FUNCTION_BLOCK FB_HDData
VAR_INPUT
	
    Alm :    BOOL ;//报警
	Wait :BOOL ;//待机
	Run :BOOL ;//运行
	XL_Wait:BOOL ;//下料等待时间
	Query:BOOL;//时间查询
	

END_VAR
VAR_OUTPUT
		STTimedata:ARRAY[0..32] OF ST_Timedata_1;

END_VAR
VAR
	
	rRun : R_TRIG;
	rAlm : R_TRIG;
	rWait : R_TRIG;
	rXL_Wait : R_TRIG;
	
	fRun: F_TRIG;
	fAlm: F_TRIG;
	fWait: F_TRIG;
    delay:BOOL ;//延时
	TON_1: TON;
	i:INT;
	K: INT;
	J: BOOL;
END_VAR

VAR_IN_OUT
     date1:INT;//查询日期
END_VAR

K:=K+1;
	IF K>499THEN
		J:=TRUE;
		K:=0;
	ELSE
		J:=FALSE;
	END_IF




///////////////运行时间/////////////////
rRun(CLK:= J , Q=> );

IF rRun.Q  AND  Run THEN
	STTimedata[system.stTime.wDay].RunTime[system.stTime.wHour]:=STTimedata[system.stTime.wDay].RunTime[system.stTime.wHour]+1;
END_IF

IF STTimedata[system.stTime.wDay].RunTime[system.stTime.wHour]> 3600 THEN
	STTimedata[system.stTime.wDay].RunTime[system.stTime.wHour]:= 3600 ;
END_IF

//IF STTimedata[system.stTime.wDay].AlmTime[system.stTime.wHour]= 0 AND STTimedata[system.stTime.wDay].WaitTime[system.stTime.wHour]= 0  AND 
   // (STTimedata[system.stTime.wDay].RunTime[system.stTime.wHour]= 3585  OR  STTimedata[system.stTime.wDay].RunTime[system.stTime.wHour]= 3586 ) THEN
	//STTimedata[system.stTime.wDay].RunTime[system.stTime.wHour]:= 3600 ;
//END_IF


///////////////待机时间///////////////
rWait(CLK:=J , Q=> );

IF rWait.Q  AND Wait THEN
	STTimedata[system.stTime.wDay].WaitTime[system.stTime.wHour]:=STTimedata[system.stTime.wDay].WaitTime[system.stTime.wHour]+1;
END_IF

IF STTimedata[system.stTime.wDay].WaitTime[system.stTime.wHour]> 3600 THEN
	STTimedata[system.stTime.wDay].WaitTime[system.stTime.wHour]:= 3600 ;
END_IF

//IF STTimedata[system.stTime.wDay].RunTime[system.stTime.wHour]= 0 AND STTimedata[system.stTime.wDay].AlmTime[system.stTime.wHour]= 0  AND 
  //   (STTimedata[system.stTime.wDay].RunTime[system.stTime.wHour]= 3585  OR  STTimedata[system.stTime.wDay].RunTime[system.stTime.wHour]= 3586 )  THEN
//	STTimedata[system.stTime.wDay].WaitTime[system.stTime.wHour]:= 3600 ;
//END_IF


////////////////报警时间///////////////
rAlm(CLK:=J , Q=> );

IF rAlm.Q AND Alm THEN
	STTimedata[system.stTime.wDay].AlmTime[system.stTime.wHour]:=STTimedata[system.stTime.wDay].AlmTime[system.stTime.wHour]+1;
END_IF

IF STTimedata[system.stTime.wDay].AlmTime[system.stTime.wHour]> 3600 THEN
	STTimedata[system.stTime.wDay].AlmTime[system.stTime.wHour]:= 3600 ;
END_IF

//IF STTimedata[system.stTime.wDay].RunTime[system.stTime.wHour]= 0 AND STTimedata[system.stTime.wDay].WaitTime[system.stTime.wHour]= 0  AND
 ////   (STTimedata[system.stTime.wDay].RunTime[system.stTime.wHour]= 3585  OR  STTimedata[system.stTime.wDay].RunTime[system.stTime.wHour]= 3586 ) THEN
//	STTimedata[system.stTime.wDay].AlmTime[system.stTime.wHour]:= 3600 ;
//END_IF

////////////////下料等待托盘时间///////////////
rXL_Wait(CLK:=J, Q=> );

IF rXL_Wait.Q AND XL_Wait THEN
	STTimedata[system.stTime.wDay].XLWaitTime[system.stTime.wHour]:=STTimedata[system.stTime.wDay].XLWaitTime[system.stTime.wHour]+1;
END_IF

//数据查询
IF Query THEN
	delay:=TRUE;
END_IF

TON_1(IN:= , PT:=T#60S , Q=> , ET=> );
IF delay THEN
		  IF NOT TON_1.Q THEN
			  TON_1.IN:=TRUE;
		  ELSE	
			  delay:=FALSE;
			  date1:=system.stTime.wDay;
		  END_IF	 
ELSE	
	 TON_1.IN:=FALSE;
END_IF


IF NOT delay THEN
STTimedata[32]:=STTimedata[system.stTime.wDay];
ELSE
STTimedata[32]:=STTimedata[date1];
END_IF

//数据清零
IF (system.stTime.wMonth=2 AND  system.stTime.wDay=28 )   OR
    ((system.stTime.wMonth=4 OR system.stTime.wMonth=6 OR system.stTime.wMonth=9 OR system.stTime.wMonth=11) AND system.stTime.wDay=30 )   OR
	((system.stTime.wMonth=1 OR  system.stTime.wMonth=3 OR system.stTime.wMonth=5 OR system.stTime.wMonth=7 OR system.stTime.wMonth=8 OR system.stTime.wMonth=10 OR system.stTime.wMonth=12) AND  system.stTime.wDay=31)  AND
    system.stTime.wHour=23 AND  system.stTime.wMinute=59 AND system.stTime.wSecond =59 THEN
	FOR i:=0 TO 32  DO
	MEMSET(ADR(STTimedata[i]),0,SIZEOF(STTimedata[i]));	
	END_FOR
END_IF

END_FUNCTION_BLOCK

(* stored: Version 1.1.0.1, ProductVersion 3.1.4024.12
   POU FB_HDData: Id {ac0a5715-ea7f-4b1b-aab9-9f16f634e643}, SpecialFunc None *)
